{attribute addProperty BoxType "EK1541-0000-0016"}
{attribute addProperty Id "IDAT %I*ID_90FEAF081620WcStateAT %I*WcState_98A4DF7520.250InfoDataAT %I*InfoData_192954DE1620"}
{attribute addProperty CRC "1114059904"}
{attribute addProperty SizeInBites "34"}
{attribute addProperty SizeInBytes "4.25"}
TYPE EK1541_963BF4D7 :
STRUCT
	{attribute addProperty Name "ID"}
	ID : ID_90FEAF08;
	{attribute addProperty Name "WcState"}
	WcState : WcState_98A4DF75;
	{attribute addProperty Name "InfoData"}
	InfoData : InfoData_192954DE;
END_STRUCT
END_TYPE

(* stored: Version 1.2.0.0, ProductVersion 3.1.4024.9
   DUT EK1541_963BF4D7: Id {d0db7aeb-6b70-4f07-a36e-ad7ad99052d3} *)
